VAR_INPUT
	in_max_Velo				: REAL;						(*	maximale Geschwindigkeit - Anwendereinheit z.B. xx mm/s *)
	in_Reglersperre			: BOOL;						(*  Software-Freigabe für die Achse  *)
	in_Freigabe				: BOOL;						(*  Freigabe JogMode und Positionieren *)
	in_Reset				: BOOL;						(*  Achs Reset  *)
	in_Hand					: BOOL;						(*  Handbetrieb  *)
	in_Auto					: BOOL;						(*  Automatikbetrieb  *)
	in_Auto_Override		: INT;						(*  in %  *)
	in_PosFenster			: REAL;						(*  Positionsfenster Achse in Position  *)
	in_Ref_pos				: REAL;						(*  Referenz-Wert der gesetzt werden soll  *)
	in_Bremse_PassQuitt		: BOOL;						(*	Passwort geschützes Bit aus der Visu zum Quittieren des Bremsentests, wenn der Test ..mal fehlgeschlagen ist	*)
	in_Endschalter_Min		: BOOL;						// AF - Reglerfreigabe für Fahrt negativ
	in_Endschalter_Max		: BOOL;						// AF - Reglerfreigabefür Fahrt positiv
	in_Normal_Drehmoment	: REAL := 100.0;			// AF - Drehmoment für den normalen Betrieb
END_VAR
VAR_OUTPUT
	out_ist_pos					: REAL;						(*  aktuelle ist Position  *)
	out_in_pos					: BOOL;						(*  Achse in Position (Soll=IST + - Positionsfenster) *)
	out_ziel_pos				: REAL;						(* aktuelle Zielposition *)
	out_nicht_ref				: BOOL;						(*  Achse ist nicht referenziert  *)
	out_bremse					: BOOL;						(*  Bremse lösen *)
	out_Achs_Status				: ST_AxisStatus;			(* 	aktueller Achsstatus *)
	out_Achs_Error				: BOOL;						(*  Achs Fehler *)
	out_Achs_ErrorID			: DINT;						(*  Achs Fehler ID *) 
	out_FB_Error				: BOOL;						(*  FB Fehler - intern *)
	out_FB_ErrorID				: DWORD;					(*  FB Fehler ID - intern *) 
	out_Bremsentest_Fehler		: BOOL;						(*	Bremsentestfehlerhaft *)
	out_Bremsentest_Fehler_3	: BOOL;						(*	Bremsentestfehlerhaft mehr als 3 mal fehlgeschlagen, Instandhalter informieren*)
	out_Bremsentest_Status		: DINT;						(*	0=alles ok, 1=Haltemoment zu gering, 2=Öffnungstest fehlerhaft, 3=...  *) 
	out_Bremsentest_notwendig	: BOOL;                       
	
END_VAR
VAR_IN_OUT
	inout_NC				: AXIS_REF;					(*  Schnittstelle zwischen der SPS und der NC  *)												
	inout_rexroth			: DUT_PD_InOut_Achsen;		(*  Schnittstelle zwischen der SPS und dem Regler  *)												
	inout_service			: DUT_Achse_Service;		(*  Eingangs-Variablen für den Servicebetrieb	 *)
	inout_Ref_start			: BOOL;						(*  Achse start referenzieren  *)
	inout_Auto_pos			: REAL;						(*  Auto Sollwert *)
	inout_Auto_start		: BOOL;						(*  Achse start Positionieren *)
	inout_Auto_stop			: BOOL;						(*  Achse stopp Positionieren *)
	inout_Bremsentest_Start	: BOOL;						(*	Bremsentest starten *)
END_VAR

VAR
	FB_ReadPos				: MC_ReadActualPosition;	(*  Aktuelle Istposition auslesen *)
	FB_ReadErrorID			: MC_ReadAxisError;			(*  FehlerID der Achse auslesen  *)
	FB_ReadStatus			: MC_ReadStatus;
	FB_POWER				: MC_POWER;					(*  Leistung ein-/ausschalten  *)
	FB_RESET				: MC_RESET;					(*  Achse resetten *)
	FB_Stop					: MC_Halt;					(*  Achse anhalten  *)
	FB_Jog					: MC_Jog;					(*  Achse tippen  *)
	FB_Move					: MC_MoveAbsolute;			(*  Achse positionieren  *)
	FB_Move_Seq_1			: MC_MoveAbsolute;
	FB_Move_Seq_2			: MC_MoveAbsolute;
	FB_Read_Parameter		: MC_ReadParameterSet;
	FB_Set_Position			: MC_SetPosition;
	FB_SoeReset				: Tc2_MC2_Drive.FB_SoEReset;
	start_seq				: BOOL;						(*  Start Merker Pos1<-> Pos 2 *)
	ton_verweil				: ton;
	ton_verzoegert			: tof;
	temp_in_pos_plus		: BOOL;
	temp_in_pos_minus		: BOOL;
	verz_reset				: ton;
	fl_start				: R_trig;					(* Start als Flanke auswerten und den Zähler erhöhen *)
	bremsentest_ver			: ton;						(* Verzögerungszeit zum Auswerten *)
	AnzahlVersuche			: INT;
	Achsparameter			: ST_AxisParameterSet;
END_VAR

// ***** Achs Status aktualisieren *******************************************************************************************
	//************************************************************************************************************************
	inout_NC();

	out_Achs_Status	:= FB_ReadStatus.Status;
	out_Achs_Error	:= FB_ReadErrorID.AxisErrorID > 0;

	IF out_Achs_Error 
		OR out_FB_Error
		OR in_reset
	THEN
		inout_Auto_start:=FALSE;
		inout_Auto_stop:=FALSE;
	END_IF
	
	if not inout_rexroth.S0145_steuerword.5 then
		inout_rexroth.S0092_drehmoment_grenzwert := REAL_TO_UINT(in_Normal_Drehmoment * 10);
	end_if
// ***** Aktuelle Zielposition ***********************************************************************************************
	//************************************************************************************************************************
	IF inout_nc.Status.Moving
	THEN
		out_ziel_pos := LREAL_TO_REAL(inout_NC.NcToPlc.TargetPos);
	ELSIF in_auto
		AND inout_auto_start
	THEN
		out_ziel_pos := inout_Auto_pos;
	ELSIF in_hand
		AND inout_service.betriebsart = 2				
			AND inout_service.plus_start
	THEN
		out_ziel_pos := inout_service.sollpos_hand;	
	END_IF	
	
// Freigabe positionieren ****************************************************************************************************
	//************************************************************************************************************************
	IF NOT in_Freigabe
	THEN
		inout_Auto_start 	:= FALSE;
		FB_Move.Execute		:= FALSE;
	END_IF	
	
// ***** Bremsentest starten *************************************************************************************************
	//************************************************************************************************************************
	out_Bremsentest_notwendig:= inout_rexroth.P0539_status_bremse.8; (* P-0-0539.8, Status Zeitintervall des Bremsentests  *)
	inout_rexroth.S0145_steuerword.2 := inout_Bremsentest_Start	(* P-0-0541, C2100 Kommando Haltesystemüberwachung *)
											AND inout_NC.Status.NotMoving;
	fl_start(clk:=inout_Bremsentest_Start);
	IF fl_start.q
	THEN
		AnzahlVersuche:=AnzahlVersuche+1;	
	END_IF
	
		// ***** Bremsentest Zeitverzögert auswerten *********************************************************************************	
			// ***********************************************************************************************************************
			bremsentest_ver(IN:=inout_rexroth.S0145_steuerword.2, pt:= T#4S);
			
		// ***** Bremsentest iO ******************************************************************************************************
			// ***********************************************************************************************************************
			IF bremsentest_ver.Q
				AND inout_rexroth.P0539_status_bremse.1 (* P-0-0539.1 - Status der Haltebremsenüberwachung *)
				AND inout_rexroth.P0539_status_bremse.2 (* P-0-0539.2 - Prüfstatus "Bremsenöffnung"  *)
				AND inout_rexroth.P0539_status_bremse.3 (* P-0-0539.3 - Prüfstatus "Haltemoment"  *)
			THEN
				inout_rexroth.S0145_steuerword.2:=FALSE;
				inout_Bremsentest_Start:=FALSE;
				AnzahlVersuche:=0;
				out_Bremsentest_Status:=0;
			END_IF
		// ***** Test niO und einen Fehler ausgeben ********************************************************************************** 
			// ***********************************************************************************************************************
			IF  bremsentest_ver.Q
					AND NOT inout_rexroth.P0539_status_bremse.2 (* P-0-0539.2 - Prüfstatus "Bremsenöffnung"  *)
			THEN
				out_Bremsentest_Status:=0;
				inout_Bremsentest_Start:=FALSE;
			END_IF
		
			IF  bremsentest_ver.Q
					AND NOT inout_rexroth.P0539_status_bremse.3 (* P-0-0539.3 - Prüfstatus "Haltemoment"  *)
			THEN
				out_Bremsentest_Status:=0;
				inout_Bremsentest_Start:=FALSE;
			END_IF
			
			IF out_Bremsentest_Status<>0
			THEN
				out_Bremsentest_Fehler:=TRUE;
				ELSE
					out_Bremsentest_Fehler:=FALSE;
			END_IF
		// ***** Quttierung nach einem Fehler ****************************************************************************************
			// ***********************************************************************************************************************
			IF AnzahlVersuche>=4
			THEN
				out_Bremsentest_Fehler_3:=TRUE;
			END_IF
			IF (in_Bremse_PassQuitt 
					OR (AnzahlVersuche<4))
				AND in_Reset
			THEN
				IF in_Bremse_PassQuitt
					AND AnzahlVersuche>=4  
				THEN
					AnzahlVersuche:=0;
				END_IF
				out_Bremsentest_Fehler_3:=FALSE;
				out_Bremsentest_Status:=0;
				inout_Bremsentest_Start:=FALSE;
			END_IF
		
// ***** Hand Betriebsart /Geschwindigkeit zurücksetzen***********************************************************************
	//************************************************************************************************************************
	IF NOT in_Hand
	THEN
		inout_service.betriebsart	:= 0;
		inout_service.override		:= 0;
	END_IF

// ***** Sollposition / Geschwindigkeit umkopieren ***************************************************************************
	//************************************************************************************************************************
	IF in_hand
	THEN
		FB_Move.Position		:= inout_service.sollpos_hand;
		FB_Power.Override		:= INT_TO_LREAL(inout_service.override);
		FB_Move.Velocity		:= in_max_velo;
		FB_Jog.Velocity			:= in_max_velo;
		fb_Move_seq_1.Velocity 	:= in_max_velo;
		fb_Move_seq_2.Velocity 	:= in_max_velo;
		fb_Move_seq_1.Position	:= inout_service.sollpos_hand;
		fb_Move_seq_2.Position	:= inout_service.pos_2;
		
		inout_rexroth.S0145_steuerword.5 := FALSE;
	ELSE
		FB_Move.Position		:= inout_Auto_pos;
		FB_Power.Override		:= INT_TO_LREAL(in_Auto_Override);
		FB_Move.Velocity		:= in_max_velo;
		FB_Jog.Velocity			:= 0.0;
	END_IF
	
	
// ***** Reset ***************************************************************************************************************
	//************************************************************************************************************************
	inout_rexroth.S0145_steuerword.0:=in_Reset;	// S-0-0099 - C0500 Reset Zustandsklasse 1 l

	FB_SoeReset(Axis := inout_NC, Execute := in_Reset OR FB_SoeReset.Busy);

	IF in_Reset
		AND (out_FB_Error
		OR out_Achs_Error) 
		OR ( in_Hand
				AND inout_service.betriebsart=0
				AND inout_service.minus_stop ) 
	THEN
		FB_Reset.Execute	:= inout_NC.NcToPlc.CoupleState <> 3; // Achse ist kein Slave
		FB_Stop.Execute		:= FALSE;
		FB_Move.Execute		:= FALSE;
		out_FB_Error		:= FALSE;
		out_FB_ErrorID		:= 0;
	END_IF

	verz_reset(	in:= FB_Reset.Execute,
				pt:= T#200MS);
	IF verz_reset.Q
	THEN
		FB_Reset.Execute := FALSE;
	END_IF

// ***** Achse stoppen *******************************************************************************************************
	//************************************************************************************************************************
	IF (in_Hand
			AND inout_service.minus_stop
			AND inout_service.betriebsart <> 1)
		OR inout_Auto_stop
		OR (NOT in_Freigabe
			AND inout_NC.Status.Moving
			AND inout_NC.NcToPlc.CoupleState <> 3) // Achse ist keine Slave Achse
		OR FB_Move.CommandAborted
		OR FB_Move.Error
		OR out_Achs_Error 
	THEN
		FB_STOP.Execute				:= TRUE;
		FB_Move.Execute				:= FALSE;
		start_seq 					:= FALSE;
		inout_service.plus_start 	:= FALSE;	
	END_IF                             
                                       
	IF (FB_STOP.Execute                
		AND FB_STOP.Done)              
	THEN                               
		inout_Auto_stop				:= FALSE;
		FB_STOP.Execute				:= FALSE;
		inout_service.minus_stop  	:= FALSE;
	END_IF

// ***** Referenzieren *******************************************************************************************************
	//************************************************************************************************************************
// Achse referenzieren - Absolutwert setzen
	inout_rexroth.S0052_ref_pos:=TRUNC(in_Ref_pos*10000.0);
	
	inout_rexroth.S0145_steuerword.1	:= NOT FB_Power.Enable
						AND ((in_Hand
								AND inout_service.betriebsart=4
								AND inout_service.plus_start)
							OR (in_Auto
								AND inout_Ref_start));

	IF inout_service.betriebsart=4
		AND (inout_rexroth.S0052_ref_pos = TRUNC(out_ist_pos*10000.0))
	THEN
		inout_service.plus_start:=FALSE;	
	END_IF
// ***** Achse positionieren *************************************************************************************************
	//************************************************************************************************************************
	IF ((in_Hand
			AND inout_service.betriebsart = 2				
			AND inout_service.plus_start)		
		OR (in_auto
			AND inout_Auto_start))
		AND NOT FB_Move.Done
		AND NOT FB_Move.busy
		AND NOT out_Achs_Error // optimierung 01.10.2020
		AND NOT out_Bremsentest_Fehler
		AND in_Freigabe
	THEN
		FB_Move.Execute:=TRUE;	
	END_IF

	IF (FB_Move.Execute
		AND FB_Move.Done)
		OR out_Achs_Error
	THEN
		FB_Move.Execute				:=FALSE;
		inout_Auto_start			:=FALSE;
		inout_service.plus_start 	:=FALSE;
	END_IF
	
	IF inout_service.betriebsart = 2
		AND (FB_Move.Execute
		AND FB_Move.Done)
	THEN 
		FB_Move.Execute := FALSE;
	END_IF
// ***** Handbetrieb - Achse POS1<->POS 2 ************************************************************************************
	//************************************************************************************************************************
	IF  in_hand
		AND inout_service.betriebsart = 3
		AND inout_service.plus_start
	THEN 
		start_seq := TRUE;
	END_IF

// ***** Handbetrieb - Achse tippen ******************************************************************************************
	//************************************************************************************************************************
	IF in_Hand
		AND inout_service.betriebsart=1
		AND NOT FB_Jog.CommandAborted
		AND NOT FB_Jog.Error
		AND NOT out_Bremsentest_Fehler
		AND in_Freigabe
	THEN
		FB_Jog.JogForward	:= inout_service.plus_start 
								AND inout_nc.NcToPlc.ActPos < (Achsparameter.fEncSoftEndMax - in_PosFenster);
		FB_Jog.JogBackwards	:= inout_service.minus_stop
								AND inout_nc.NcToPlc.ActPos > (Achsparameter.fEncSoftEndMin + in_PosFenster);
		
		// Geschwindigkeit tippen vor den Endlagen reduzieren
			// letzer 1% des Fahrwegs
		IF (FB_Jog.JogForward 
			AND inout_nc.NcToPlc.ActPos 
				> Achsparameter.fEncSoftEndMax - ((Achsparameter.fEncSoftEndMax - Achsparameter.fEncSoftEndMin) * 0.01))
			
			OR (FB_Jog.JogBackwards
				AND inout_nc.NcToPlc.ActPos  
					< Achsparameter.fEncSoftEndMin + ((Achsparameter.fEncSoftEndMax - Achsparameter.fEncSoftEndMin) * 0.01))
					
			AND FB_Power.Override > 5
		THEN
			FB_Power.Override := 5;
			
			// letzten 5% des Fahrwegs
		ELSIF (FB_Jog.JogForward 
			AND inout_nc.NcToPlc.ActPos 
				> Achsparameter.fEncSoftEndMax - ((Achsparameter.fEncSoftEndMax - Achsparameter.fEncSoftEndMin) * 0.05))
			
			OR (FB_Jog.JogBackwards
				AND inout_nc.NcToPlc.ActPos  
					< Achsparameter.fEncSoftEndMin + ((Achsparameter.fEncSoftEndMax - Achsparameter.fEncSoftEndMin) * 0.05))
					
			AND FB_Power.Override > 10	
		THEN
			FB_Power.Override := 10;
		END_IF
	ELSE
		FB_Jog.JogForward	:= FALSE;
		FB_Jog.JogBackwards	:= FALSE;
	END_IF
	
// ***** Aufruf der FB´s  ****************************************************************************************************
	//************************************************************************************************************************
	 ACT_Achse_NC_PTP();	
				
// ***** Bremse lösen ********************************************************************************************************
	//************************************************************************************************************************
	ton_verzoegert.IN 	:= FB_ReadStatus.Status.HasJob; 
	ton_verzoegert.pt 	:= T#2S;
	ton_verzoegert();
	out_bremse			:= ton_verzoegert.Q;
	
// ***** Achse in Position ***************************************************************************************************
	//************************************************************************************************************************
	out_in_pos := FB_ReadStatus.Status.InTargetPosition
					AND ((out_ist_pos >= (inout_Auto_pos - in_PosFenster))
					AND (out_ist_pos <= (inout_Auto_pos + in_PosFenster)));
					
// ***** Achse Referenzert ***************************************************************************************************
	//************************************************************************************************************************
	out_nicht_ref:=	 inout_rexroth.S0144_statusword.0;	//NOT FB_ReadStatus.Status.Homed;

// ***** FB Fehler auswerten und ausgeben ************************************************************************************
	//************************************************************************************************************************
	IF FB_Jog.Error
		AND FB_Jog.ErrorID > 0
	THEN
		out_FB_Error	:= TRUE;
		out_FB_ErrorID	:= FB_Jog.ErrorID;
		
	ELSIF FB_Move.Error
		AND FB_Move.ErrorID>0
	THEN
		FB_Move.Execute	:= FALSE;
		out_FB_Error	:= TRUE;
		out_FB_ErrorID	:= FB_Move.ErrorID;
		
	ELSIF FB_Stop.Error
		AND FB_Stop.ErrorID>0
	THEN	
		FB_Stop.Execute	:= FALSE;
		out_FB_Error	:= TRUE;
		out_FB_ErrorID	:= FB_Stop.ErrorID;
		
	ELSIF FB_Reset.Error
		AND FB_Reset.ErrorID>0
	THEN
		FB_Reset.Execute	:= FALSE;
		out_FB_Error		:= TRUE;
		out_FB_ErrorID		:= FB_Reset.ErrorID;
	END_IF			

					
// ***** Servicetasten zurück setzen ************************************************************************************
	//************************************************************************************************************************
	IF inout_service.betriebsart <> 1
		AND inout_service.betriebsart <> 4
	THEN
		inout_service.plus_start := FALSE;				
		inout_service.minus_stop := FALSE;				
	END_IF
	
	inout_Auto_start := FALSE;

ACTION ACT_Achse_NC_PTP:
	
	FB_ReadErrorID(	Axis:=inout_NC,
					Enable:=TRUE,
					AxisErrorID=>);
	out_achs_ErrorID:= DWORD_TO_DINT(FB_ReadErrorID.AxisErrorID);	
	
	
	FB_ReadPos(		Axis:=inout_NC,
					Enable:=TRUE,
					Position=> ,
					Position=> );				
				
	out_ist_pos:=inout_service.istpos:=LREAL_TO_REAL(FB_ReadPos.Position);
	
	FB_Read_Parameter(	Parameter:= Achsparameter, 
						Axis:= inout_NC, 
						Execute:= in_Reglersperre, 
						Done=> , 
						Busy=> , 
						Error=> , 
						ErrorID=> );
			
	FB_ReadStatus(	Axis:=inout_NC,
					Enable:=TRUE);
				
	FB_Power.Enable:=in_Reglersperre AND (inout_service.betriebsart<>4	OR inout_ref_start);	
	FB_Power.Enable_Negative := FB_Power.Enable AND in_Endschalter_Min;
	FB_Power.Enable_Positive :=	FB_Power.Enable	AND in_Endschalter_Max;
				
	FB_Power(	Axis:=inout_NC,
				Enable:=,
				Enable_Positive:=,
				Enable_Negative:=,
				Override:=,
				BufferMode:=MC_Aborting,
				Options:=	);
				
	FB_Reset(	Axis:=inout_NC,
				Execute:=	);
				
	FB_Stop(	Axis:=inout_NC,
				Execute:=,
				Deceleration:=0,				(* Bei einem Wert von 0 wirkt die mit dem letzten Move-Kommando parametrierte Verzögerung *)
				Jerk:=0,						(* Bei einem Wert von 0 wirkt der mit dem letzten Move-Kommando parametrierte Ruck *)		
				BufferMode:= MC_Aborting);		 // Wichtig !!!!				
																		
	FB_Move(	Axis:=inout_NC,
				Execute:=,
				Position:=,
				Velocity:=,
				Acceleration:=0,				(* Beschleunigung, bei einem Wert von 0 wirkt die Standardbeschleunigung aus der Achskonfiguration im System Manager *)
				Deceleration:=0,				(* Verzögerung, bei einem Wert von 0 wirkt die Standardverzögerung aus der Achskonfiguration im System Manager *)
				Jerk:=0, 						(* Ruck, bei einem Wert von 0 wirkt der Standardruck aus der Achskonfiguration im System Manager *)
				BufferMode:= MC_Buffered);		
									
	FB_Jog(		Axis:=inout_NC,
				JogForward:=,
				JogBackwards:=,
				Mode:= MC_JOGMODE_STANDARD_SLOW, //MC_JOGMODE_CONTINOUS,
				Position:=,						(* nicht in diesem Mode notwendig *)
				Velocity:=,
				Acceleration:=0,				(* Beschleunigung, bei einem Wert von 0 wirkt die Standardbeschleunigung aus der Achskonfiguration im System Manager *)
				Deceleration:=0,				(* Verzögerung, bei einem Wert von 0 wirkt die Standardverzögerung aus der Achskonfiguration im System Manager *)
				Jerk:=0 );						(* Ruck, bei einem Wert von 0 wirkt der Standardruck aus der Achskonfiguration im System Manager *)

	
	ton_verweil(in:= (NOT fb_move_seq_1.active 
						AND NOT fb_move_seq_2.active
						AND inout_service.betriebsart=3),
				pt:= INT_TO_TIME(inout_service.zeit));
				
	FB_Move_Seq_1(
				Execute:= 	(start_seq 
								AND NOT fb_move_seq_2.busy 
								AND ton_verweil.Q),
				Position:= 			,
				Velocity:= 			,
				Acceleration:= ,				(* Beschleunigung, bei einem Wert von 0 wirkt die Standardbeschleunigung aus der Achskonfiguration im System Manager *)
				Deceleration:= ,			 	(* Verzögerung, bei einem Wert von 0 wirkt die Standardverzögerung aus der Achskonfiguration im System Manager *)
				Jerk:=,							(* Ruck, bei einem Wert von 0 wirkt der Standardruck aus der Achskonfiguration im System Manager *) 
				BufferMode:= MC_Buffered,
				Options:= ,
				Axis:=inout_NC,
				Done=>				,
				Busy=> 				,
				Active=> 			,
				CommandAborted=> 	,
				Error=> 			,
				ErrorID=> 			);


	FB_Move_Seq_2(
				Execute:= 		(start_seq	
								AND fb_move_seq_1.done
								AND ton_verweil.Q),
				Position:= 		,
				Velocity:= 			,
				Acceleration:= ,				(* Beschleunigung, bei einem Wert von 0 wirkt die Standardbeschleunigung aus der Achskonfiguration im System Manager *)
				Deceleration:= ,				(* Verzögerung, bei einem Wert von 0 wirkt die Standardverzögerung aus der Achskonfiguration im System Manager *)
				Jerk:= ,						(* Ruck, bei einem Wert von 0 wirkt der Standardruck aus der Achskonfiguration im System Manager *)
				BufferMode:= MC_Buffered,
				Options:= ,
				Axis:= inout_NC,
				Done=>				,
				Busy=> 				,
				Active=> 			,
				CommandAborted=> 	,
				Error=> 			,
				ErrorID=> 			);
END_ACTION

METHOD M_AutoPos : BOOL
VAR_INPUT
	SollPos		:REAL;
END_VAR
	
	// Drehmomentgrenze deaktivieren
	inout_rexroth.S0145_steuerword.5 := FALSE;

	if not inout_rexroth.S0144_statusword.6 then
		FB_Move.Options.IgnorePositionMonitoring := false;
		
		inout_Auto_pos := SollPos;
		inout_Auto_start := TRUE;
	
		IF out_in_pos 
		AND Func_InRange(IstPos := inout_NC.NcToPlc.ActPos, SollPos := inout_Auto_pos, Fenster := in_PosFenster) 
		THEN
			M_AutoPos := TRUE;
		END_IF 
		
	end_if
END_METHOD

METHOD M_AutoTorque : BOOL
VAR_INPUT
	SollPos	: REAL;
	Torque	: REAL;  // Prozentwert
END_VAR
	
	inout_rexroth.S0145_steuerword.5 := TRUE;
	if inout_rexroth.S0144_statusword.6 then
		FB_Move.Options.IgnorePositionMonitoring := true;
		inout_rexroth.S0092_drehmoment_grenzwert := REAL_TO_UINT(Torque * 10);
	
		inout_Auto_pos := SollPos;
		inout_Auto_start := TRUE;
	
		IF (out_in_pos 
		AND Func_InRange(IstPos := inout_NC.NcToPlc.ActPos, SollPos := inout_Auto_pos, Fenster := in_PosFenster))
		OR inout_rexroth.S0144_statusword.5
		THEN
			M_AutoTorque := TRUE;
		END_IF 
	
	end_if
END_METHOD

END_FUNCTION_BLOCK

// ---- SRT_Allgemein/0010_Bausteine_mitDuts/POUs/Servos_NC/FB_MasterSlaveSpeedControl.TcPOU
FUNCTION_BLOCK FB_MasterSlaveSpeedControl
VAR_INPUT
	SpeedMaster	:REAL;
	SpeedSlave1	:REAL;
	SpeedSlave2	:REAL;
	SpeedSlave3	:REAL;
	hysterese	:REAL;
	
END_VAR
VAR_OUTPUT
	speedMasterSlave_OK :BOOL;
END_VAR
VAR
	speedSlave1_OK	:BOOL;
	speedSlave2_OK	:BOOL;
	speedSlave3_OK	:BOOL;
END_VAR

IF SpeedSlave1 < SpeedMaster + hysterese
	AND SpeedSlave1 > SpeedMaster - hysterese
THEN
	speedSlave1_OK :=TRUE;
ELSE
	speedSlave1_OK :=FALSE;
END_IF

IF SpeedSlave2 < SpeedMaster + hysterese
	AND SpeedSlave2 > SpeedMaster - hysterese
THEN
	speedSlave2_OK :=TRUE;
ELSE
	speedSlave2_OK :=FALSE;
END_IF

IF SpeedSlave3 < SpeedMaster + hysterese
	AND SpeedSlave3 > SpeedMaster - hysterese
THEN
	speedSlave3_OK :=TRUE;
ELSE
	speedSlave3_OK :=FALSE;
END_IF


IF speedSlave1_OK
	AND speedSlave2_OK
	AND speedSlave3_OK
	AND speedMaster>0
THEN
	speedMasterSlave_ok := TRUE;
ELSE
	speedMasterSlave_ok := FALSE;
END_IF

END_FUNCTION_BLOCK

// ---- SRT_Allgemein/0010_Bausteine_mitDuts/POUs/Servos_NC/FB_Nc_Kanal.TcPOU
FUNCTION_BLOCK FB_Nc_Kanal
(*
	Ansteuerung eines NC-Kanals 
	Autor O.E.
	Erstellt 13.01.2022
	Version 1.0 	
*)
VAR_INPUT
	in_Kanal_Id						:UDINT;					(* NC Kanal Nummer *)
	in_Gruppe_Id					:UDINT;					(* NC Gruppennummer *)
	in_X_Id							:UDINT;					(* X-Achs Id *)
	in_Y_Id							:UDINT;					(* Y-Achs Id *)
	in_Z_Id							:UDINT;					(* Z-Achs Id *)
	in_Pfad							:STRING[80];			(* Pfad wo das NC-Programm liegr *)
	in_PName						:STRING[80];			(* Name des zubearbeitenden NC-Programms *)
	in_Override						:DINT;					(* Gesamt Override der bearbeitung 0-100%*)
	in_NcToPlc						:NCTOPLC_NCICHANNEL_REF;
END_VAR

VAR_OUTPUT
	out_PlcToNc						:PLCTONC_NCICHANNEL_REF;
	out_P_uebernommen				:BOOL;					(* vorgegebenes Programm übernommen soll=ist *)
	out_FBErr						:BOOL;
	out_FBErrId						:UDINT;
END_VAR

VAR_IN_OUT
	inout_NcReset					:BOOL;				(* Kanal Reset *)
	inout_NcGruppe_koppeln			:BOOL;				(* Achsen zu einer Gruppe zusammen fügen *)
	inout_NcStart					:BOOL;				(* NC-Ablauf starten *)
	inout_NcStopOverrideNull		:BOOL;				(* NC-Ablauf unterbrechen -Override=0 *)
	inout_NcEinzelsatzStart			:BOOL;				(* NC-Ablauf im Einzelsatzbetrieb abarbeiten *)
	inout_NcEinzelsatzWeiter		:BOOL;				(* nächster Satz *)
	inout_NcStatus					:Dut_Nc_Kanal;
	
END_VAR

VAR
	                    	
	AxTo3D			 				:CfgBuildExt3dGroup;
	AxToPTP							:CfgReconfigGroup;
	AxTo3DLoad						:BOOL;
	AxToPTPLoad						:BOOL;                  		
                            	
	Einzel							:ItpsingleBlock;
	EinzelChange					:BOOL;
	EinzelStart						:R_Trig;
	EinzelStop						:f_Trig;
	ProgAnw							:ItpLoadProgEx;
	ProgStart						:ItpStartStopEx;
	ProgReset						:ItpResetEx;
                    			
	PLoad							:BOOL;
	
	FlPGrd							:R_TRIG;
	FlPBearb						:R_TRIG;
	Pfad_PNr 	 					:STRING[80];
	FlPReset						:R_Trig;
                    	    	
	TStart							:TON;
	PStart							:R_TRIG;
                    				
	OverInit						:BOOL;
                   				
	MFuncTime						:TON;
    MFuncQuitt						:ItpResetFastMFuncEx;  
	MFuncConfirm					:ItpConfirmHsk;
	FlMFuncNoReq					:r_trig;

	PName_akt:						STRING[80];
	
	PBearb:							BOOL;
	Override						:DINT;
	Start:							BOOL;
	Stop:							BOOL;
	Untbr:							BOOL;
	Reset:							BOOL;

	 
END_VAR

//***** Info zum NCI-Ablauf *************************************************************************************
	//**********************************************************************************************************
(*
	1. Einzelachsen fehlerfrei in Grundposition
	2. Gruppe bilden / Achsen koppeln			-> CfgBuildExt3dGroup
	3. Interpreter Reset						-> ItpResetEx
	4. Programm laden							-> ItpLoadProgEx
	5. Einzelsatzbetrieb (optinal)				-> ItpSingleBlock
	6. Programm starten							-> ItpStartStopEx
	7. Warten auf M-Funktion und quittieren		-> PLCTONC_NCICHANNEL_REF.MFuncGranted
		M-Funktion steht an							-> ItpIsHskMFunc
		M_FunktionsNummer							-> ItpGetHskMFunc
	8. Gruppe auflösen / Achsen entkoppeln		-> CfgReconfigGroup
*)
//***** Kanalreset *********************************************************************************************
	//**********************************************************************************************************
	Reset:= inout_NcReset;

//***** Achsen Config ******************************************************************************************
	//**********************************************************************************************************

		IF inout_NcGruppe_koppeln
		THEN
			IF NOT inout_NcStatus.AxTo3DOk
			AND NOT AxTo3D.bErr
			THEN
				AxTo3DLoad:= TRUE;
				inout_NcStatus.AxToPTPOk:= FALSE;
			END_IF;
		ELSE
			IF NOT inout_NcStatus.AxToPTPOk
			AND NOT AxToPTP.bErr
			THEN
				AxToPTPLoad:= TRUE;
				inout_NcStatus.AxTo3DOk:= FALSE;
			END_IF;
		END_IF;

	// Achsen in 3D Gruppe uebergeben 
	AxTo3D	(	nGroupId		:=in_Gruppe_Id,
				nXAxisId		:=in_X_Id,
				nYAxisId		:=in_Y_Id,
				nZAxisId		:=in_Z_Id,
				nQ1AxisId		:=0,
				nQ2AxisId		:=0,
				nQ3AxisId		:=0,
				nQ4AxisId		:=0,
				nQ5AxisId		:=0,
				bExecute		:=AxTo3DLoad,
				tTimeOuT		:=T#1S,				
				bErr			=>,
				nErrId			=>,);


	IF AxTo3D.bBusy THEN
		inout_NcStatus.AxTo3Dok	:= TRUE;
		AxTo3DLoad			:= FALSE;
	END_IF;

	IF AxTo3D.bErr THEN
		inout_NcStatus.AxTo3Dok	:= FALSE;
	END_IF;

	// Achsen zurueck in PTP 
	AxToPTP(nGroupId		:=in_Gruppe_Id,
			bExecute		:=AxToPTPLoad,
			tTimeOuT		:=T#1S);

	IF AxToPTP.bBusy THEN
		inout_NcStatus.AxToPTPok	:= TRUE;
		AxToPTPLoad			:= FALSE;
	END_IF;

	IF AxToPTP.bErr THEN
		inout_NcStatus.AxToPTPok	:= FALSE;
	END_IF;
	
//***** Aktuelles NC-Programm laden ***************************************************************************
	//**********************************************************************************************************
	PName_akt		:=DWORD_TO_STRING (in_NcToPlc.LoadedProg);
	
	// NC-Programm laden 
	IF in_PName <> PName_akt
		AND NOT Reset
		AND NOT ProgAnw.bBusy 
		AND in_PName <>''
	THEN
		PLoad:=TRUE;
		ELSE
			PLoad:=FALSE;
	END_IF;

	Pfad_PNr := CONCAT (in_Pfad, in_PName) ;
	Pfad_PNr := CONCAT (Pfad_PNr,'.NC') ;

	ProgAnw (sNciToPlc	:=in_NcToPlc,
			sPrg		:=Pfad_PNr,
			nLength		:=INT_TO_UDINT((LEN(Pfad_PNr))),
			bExecute	:=PLoad,
			tTimeOuT	:=T#10S,				
			bErr		=>,
			nErrId		=>);

	IF ProgAnw.bBusy 
	THEN
		PLoad			:= FALSE;
	END_IF;

	// Ueberpruefung Grundstellung / Bearbeitungsprogramm geladen 
	PBearb	:=(in_PName = PName_akt);
	// Nach dem laden des Programmes muß ein Reset durchgefuehrt werden 
	FlPBearb (CLK:=PBearb);

	IF FlPGrd.Q
	OR FlPBearb.Q
	THEN
		Reset:= TRUE;
	END_IF;

	out_P_uebernommen:= in_PName = PName_akt;
//***** NC Err *************************************************************************************************
	//**********************************************************************************************************
	inout_NcStatus.Err	:=  in_NcToPlc.ItpState= Tc2_NCI.NCI_INTERPRETER_ABORTED
					 OR in_NcToPlc.ErrorCode<> 0;

//***** NC Aktiv ***********************************************************************************************
	//**********************************************************************************************************
	inout_NcStatus.Aktiv	:= in_NcToPlc.ItpState > Tc2_NCI.NCI_INTERPRETER_READY
					AND NOT inout_NcStatus.Err;

//***** NC Ready ***********************************************************************************************
	//**********************************************************************************************************
	IF in_NcToPlc.ItpState = Tc2_NCI.NCI_INTERPRETER_READY
	THEN
		inout_NcStatus.Ready:= TRUE;
	END_IF

	IF in_NcToPlc.ItpState = Tc2_NCI.NCI_INTERPRETER_IDLE
		OR inout_NcStatus.Err
		OR inout_NcStatus.Aktiv
	THEN
		inout_NcStatus.Ready:= FALSE;
	END_IF
//***** NC Run *************************************************************************************************
	//**********************************************************************************************************
	inout_NcStatus.Run	:= in_NcToPlc.ItpState = Tc2_NCI.NCI_INTERPRETER_RUNNING;
				
//***** Einzelsatzbetrieb **************************************************************************************
	//**********************************************************************************************************
	EinzelStart(clk:=inout_NcEinzelsatzStart);
	EinzelStop(clk:=inout_NcEinzelsatzStart);
	
	IF EinzelStart.q 
		AND NOT inout_NcStart
		AND in_NcToPlc.ItpState = Tc2_NCI.NCI_INTERPRETER_READY
	THEN
		//  ItpSingleBlockOff   	:= 0 		-> Einzelsatz aus
		//	ItpSingleBlockNck   	:= 1 		-> Einzelsatz im NC-Kern
		//	ItpSingleBlockIntp  	:= 16#4000	-> Einzelsatz im Interpreter
		Einzel.nMode:= ItpSingleBlockIntp  ;
		EinzelChange:=TRUE;
	END_IF

	IF EinzelStop.Q
	THEN 
		Einzel.nMode:=ItpSingleBlockOff;
		EinzelChange:=TRUE;
	END_IF
		
	Einzel(sNciToPlc			:= in_NcToPlc,
			bExecuteModeChange	:= EinzelChange,
			bTriggerNext		:= inout_NcEinzelsatzWeiter);
		
	IF Einzel.bBusy
	THEN
		EinzelChange:=FALSE;
	END_IF	
//***** NC Start/Stop Programm *********************************************************************************
	//**********************************************************************************************************
	TStart.IN	:=inout_NcStart 
					AND inout_NcStatus.AxTo3DOk
					AND NOT EinzelChange;
	TStart(PT	:=T#50ms);

	PStart (CLK:=TStart.Q);

	IF PStart.Q
	THEN
		Start:=TRUE;
	END_IF

	IF NOT  inout_NcStart
		OR 	inout_NcStatus.Aktiv
	THEN
		Start:=FALSE;
	END_IF 

	IF NOT inout_NcGruppe_koppeln
		AND in_NcToPlc.ItpState = Tc2_NCI.NCI_INTERPRETER_RUNNING
	THEN
		Stop:=TRUE;
		Reset:=TRUE;
	END_IF


	IF in_NcToPlc.ItpState <> Tc2_NCI.NCI_INTERPRETER_RUNNING
	THEN
		Stop:=FALSE;
	END_IF

	ProgStart(sNciToPlc		:=in_NcToPlc,
				bStart		:=Start,
				bStop		:=Stop,
				tTimeOut	:=T#1S,				
				bErr		=>,
				nErrId		=>);

	IF ProgStart.bBusy
	THEN
		Start:= FALSE;
		Stop:= FALSE;
	END_IF;

//***** NC Reset Programm **************************************************************************************
	//**********************************************************************************************************
	IF  in_NcToPlc.ItpState = Tc2_NCI.NCI_INTERPRETER_READY
		AND in_NcToPlc.ErrorCode = 0
	THEN
		Reset:= FALSE;
	END_IF;

	ProgReset(nChnId	:=in_Kanal_Id,
				nGrpId	:=in_Gruppe_Id,	
				bExecute:=Reset,
				tTimeOut:=T#1S,				
				bErr		=>,
				nErrId		=>);

	Reset:= FALSE;

//***** Kanal Override *****************************************************************************************
	//**********************************************************************************************************
	IF NOT OverInit
	THEN
		in_Override	:=1000000;	(* Init 100% *)
		OverInit	:=TRUE;
	ELSE
		Override:=in_Override*10000;
	END_IF;

	out_PlcToNc.ChnAxesOvr 		:=DINT_TO_UDINT(Override);

	Untbr					:=inout_NcStopOverrideNull;

	IF Untbr
	THEN
		out_PlcToNc.ChnAxesOvr:=0; (* 0% *)
	END_IF;

//***** M-Befehle **********************************************************************************************
	//**********************************************************************************************************
	inout_NcStatus.MFuncReq:=ItpIsHskMFunc(in_NcToPlc);
	inout_NcStatus.MFuncNr:=ItpGetHskMFunc(in_NcToPlc);
	 
 
	MFuncTime(IN:=(inout_NcStatus.MFuncReq), PT:=T#100MS);

	IF MFuncTime.Q
		AND inout_NcStatus.MFuncQuitt 
		AND (inout_NcStatus.MFuncNr=inout_NcStatus.MFuncQuittNr)
	THEN
		out_PlcToNc.MFuncGranted:=1;
		ELSE
			out_PlcToNc.MFuncGranted:=0;			
	END_IF

	FlMFuncNoReq(clk:=NOT inout_NcStatus.MFuncReq);															
	IF FlMFuncNoReq.Q
	THEN  		
		inout_NcStatus.MFuncQuitt:=FALSE;														
	END_IF
	
//***** Fehler ausgeben ****************************************************************************************
	//**********************************************************************************************************

	IF ProgAnw.bErr
	THEN
		out_FBErr:=TRUE;
		out_FBErrId:=ProgAnw.nErrId;
	END_IF
	
	IF ProgStart.bErr
	THEN
		out_FBErr:=TRUE;
		out_FBErrId:=ProgStart.nErrId;
	END_IF

	IF AxTo3D.bErr
	THEN
		out_FBErr:=TRUE;
		out_FBErrId:=AxTo3D.nErrId;
	END_IF

	IF AxToPTP.bErr
	THEN
		out_FBErr:=TRUE;
		out_FBErrId:=AxToPTP.nErrId;
	END_IF

	IF ProgReset.bErr
	THEN
		out_FBErr:=TRUE;
		out_FBErrId:=ProgReset.nErrId;
	END_IF
	
//*****************************************************************************************************
	//**********************************************************************************************************
	FlPReset(clk:=in_NcToPlc.ItpState = Tc2_NCI.NCI_INTERPRETER_READY);
	IF FlPReset.Q
		OR inout_NcReset
	THEN
		inout_NcGruppe_koppeln			:=
		inout_NcStart					:=
		inout_NcStopOverrideNull		:=
		inout_NcEinzelsatzStart			:=
		inout_NcEinzelsatzWeiter		:=
		inout_NcStatus.MFuncQuitt		:=FALSE;
		inout_NcStatus.MFuncQuittNr		:=0;
	
		IF NOT ProgAnw.bErr
			AND NOT ProgStart.bErr
			AND NOT AxTo3D.bErr
			AND NOT AxToPTP.bErr
			AND NOT ProgReset.bErr
		THEN
			out_FBErr					:=FALSE;
			out_FBErrId					:=0;
		END_IF

			inout_NcReset				:=FALSE;		
		
	END_IF

END_FUNCTION_BLOCK

// ---- SRT_Allgemein/0010_Bausteine_mitDuts/POUs/Zaehler/FB_Laufzeit.TcPOU
FUNCTION_BLOCK FB_Laufzeit
VAR_INPUT
    inAktiv				: BOOL;		(* Betriebsstatus, 1 = aktiv, 0 = inaktiv *)
END_VAR

VAR_OUTPUT
    outLetzeteLaufzeit	: REAL;		(* letzte Laufzeit in Sekunden *)	
END_VAR

VAR_IN_OUT
    inoutGesamtLaufzeit	: REAL;		(* Gesamt Laufzeit in Minuten *)	
END_VAR

VAR
	t500msAn			: ton;
	t500msAus			: tof;
	t500ms				: BOOL;
	fl_start			: r_trig;
	fl_stop				: f_trig;
	zaehler				: UDINT;
END_VAR

(* Blinktakt *)
	t500msAn(IN:=NOT t500msAus.Q , PT:=T#500MS);
	t500msAus(IN:=t500msAn.Q , PT:=T#500MS , Q=>t500ms);
	
(* Start *)
	fl_start(CLK:=t500ms AND inAktiv);
	IF fl_start.Q
	THEN
		zaehler:=zaehler+1;
	END_IF
	
(* Zählwert auswertent *)
	fl_stop(CLK:=inAktiv);
	IF fl_stop.Q
	THEN
		outLetzeteLaufzeit:=	TO_REAL (zaehler);
		inoutGesamtLaufzeit:= 	inoutGesamtLaufzeit + (TO_REAL (zaehler)/60);
	END_IF

(* Initialisierung des internen Zählers *)
	IF NOT inAktiv
	THEN
		zaehler:=0;
	END_IF

END_FUNCTION_BLOCK

// ---- SRT_Allgemein/0010_Bausteine_mitDuts/POUs/Zaehler/FB_SpindelInBearbeitung.TcPOU
FUNCTION_BLOCK FB_SpindelInBearbeitung
VAR_INPUT
	inStart				:BOOL;	
	inAktiveSpindeln	:ARRAY[1..16] OF BOOL; 		// aktive Spindeln im Bohrvorgang
END_VAR
VAR_IN_OUT
	inoutSpindel		:ARRAY[1..16] OF UDINT; 	// Anzahl wie oft eine Spindel benutzt wurde
END_VAR
VAR
	a					: INT:=1;
	fl_start			: r_trig;	
END_VAR

	fl_start(CLK:=inStart);
	IF fl_start.Q
	THEN
		FOR a:=1 TO 16 DO
			IF inAktiveSpindeln[a]
			THEN
				inoutSpindel[a]:=inoutSpindel[a]+1;
			END_IF
		END_FOR		
	END_IF

END_FUNCTION_BLOCK

// ---- SRT_Allgemein/Bus/Busdiagnose.TcPOU
FUNCTION_BLOCK Busdiagnose
VAR_INPUT
			
	
END_VAR
VAR_OUTPUT
	
END_VAR
VAR_IN_OUT
Bus:DUT_Busdiagnose;
END_VAR
VAR
{attribute 'tc_no_symbol'}
StatesLesen : FB_ecGetAllSlaveStates;
{attribute 'tc_no_symbol'}
AddressenLesen : FB_EcGetConfSlaves;
{attribute 'tc_no_symbol'}
TopologieLesen: FB_EcGetSlaveTopologyInfo;
{attribute 'tc_no_symbol'}
AnzahlEtherCatDevices: FB_EcGetSlaveCount;
{attribute 'tc_no_symbol'}
Slaveslesen: FB_EcGetScannedSlaves;
{attribute 'tc_no_symbol'}
States	 : ARRAY [0..ec_Max_Slaves] OF ST_EcSlaveState;
{attribute 'tc_no_symbol'}
StatesAlt	 : ARRAY [0..ec_Max_Slaves] OF ST_EcSlaveState;
{attribute 'tc_no_symbol'}
Config	 : ARRAY [0..ec_Max_Slaves] OF ST_EcSlaveConfigData;
{attribute 'tc_no_symbol'}
Topology	 : ARRAY [0..ec_Max_Slaves] OF ST_TopologyDataEx;
{attribute 'tc_no_symbol'}
Slaves	 : ARRAY [0..ec_Max_Slaves] OF ST_EcSlaveScannedData;
{attribute 'tc_no_symbol'}
lesen :BOOL;
{attribute 'tc_no_symbol'}

{attribute 'tc_no_symbol'}
busy:BOOL;
{attribute 'tc_no_symbol'}
error:BOOL;
{attribute 'tc_no_symbol'}
errorId: UDINT;
{attribute 'tc_no_symbol'}
Slave: UINT;

{attribute 'tc_no_symbol'}	
busy2:BOOL;
{attribute 'tc_no_symbol'}
error2:BOOL;
{attribute 'tc_no_symbol'}
errorID2: UDINT;
{attribute 'tc_no_symbol'}
Slaves2: UINT;

{attribute 'tc_no_symbol'}	
busy3:BOOL;
{attribute 'tc_no_symbol'}
error3:BOOL;
{attribute 'tc_no_symbol'}
errorID3: UDINT;
{attribute 'tc_no_symbol'}
Slaves3: UINT;

{attribute 'tc_no_symbol'}	
busy4:BOOL;
{attribute 'tc_no_symbol'}
error4:BOOL;
{attribute 'tc_no_symbol'}
errorID4: UDINT;
{attribute 'tc_no_symbol'}
Slaves4: UINT;

{attribute 'tc_no_symbol'}	
busy5:BOOL;
{attribute 'tc_no_symbol'}
error5:BOOL;
{attribute 'tc_no_symbol'}
errorID5: UDINT;
{attribute 'tc_no_symbol'}
Slaves5: UINT;

{attribute 'tc_no_symbol'}	
zyklen : INT;
{attribute 'tc_no_symbol'}
i: UDINT;
{attribute 'tc_no_symbol'}	
AnzahlFehler :UINT;
END_VAR



AnzahlEtherCatDevices(
	sNetId:= F_CreateAmsNetId(nIds:=  bus.AmsNetId), 
	bExecute:= lesen, 
	tTimeout:=T#500MS , 
	bBusy=> busy4 , 
	bError=> error4, 
	nErrId=>errorID4 , 
	nSlaves=> Bus.AnzahlTeilnehmer);

StatesLesen(
	sNetId:= F_CreateAmsNetId(nIds:=  bus.AmsNetId),
	pStateBuf:= ADR(States), 
	cbBufLen:= SIZEOF(States), 
	bExecute:= lesen, 
	tTimeout:= T#500MS, 
	bBusy=>busy , 
	bError=> error, 
	nErrId=> errorId, 
	nSlaves=> Slave
 );
 
 AddressenLesen(
	sNetId:=F_CreateAmsNetId(nIds:=  bus.AmsNetId), 
	pArrEcConfSlaveInfo:= ADR(Config) , 
	cbBufLen:= SIZEOF(Config), 
	bExecute:= lesen, 
	tTimeout:=  T#500MS, 
	bBusy=> busy2, 
	bError=> error2,
	nErrorId=> errorID2, 
	nSlaves=> Slaves2);
	
TopologieLesen(
	sNetId:= F_CreateAmsNetId(nIds:=  bus.AmsNetId), 
	pAddrBuf:= ADR(Topology) , 
	cbBufLen:= SIZEOF(Topology), 
	bExecute:= lesen, 
	tTimeout:= T#500MS, 
	bBusy=> busy3, 
	bError=> error3,
	nErrId=> errorID3, 
	nSlaves=> Slaves3);
	
	Slaveslesen(sNetId:= F_CreateAmsNetId(nIds:=  bus.AmsNetId), 
	pArrEcScannedSlaveInfo := ADR(slaves) , 
	cbBufLen:= SIZEOF(slaves), 
	bExecute:= lesen, 
	tTimeout:= T#500MS, 
	bBusy=> busy5, 
	bError=> error5,
	nErrorId=> errorID5, 
	nSlaves=> Slaves5);
	
	zyklen := zyklen + 1;
	
	IF zyklen >= 100 THEN
		zyklen := 0;
		lesen := NOT lesen;
	END_IF
	
	IF Bus.AnzahlTeilnehmer > SIZEOF(Bus.Daten) THEN
		Bus.AnzahlTeilnehmer := SIZEOF(Bus.Daten);
		END_IF
		
	IF  Bus.AnzahlTeilnehmer > 0 AND lesen AND Config[0].sType <> ''
AND NOT busy
AND NOT busy2
AND NOT busy3
AND NOT busy4
//AND NOT busy5

 THEN
		FOR i := 0 TO  Bus.AnzahlTeilnehmer-1 DO
			
			Bus.Daten[i].adresse := Config[i].nAddr;
			Bus.Daten[i].deviceState := States[i].deviceState;
			Bus.Daten[i].linkState := States[i].linkState;
			Bus.Daten[i].Name := Config[i].sName;
			Bus.Daten[i].PortA := Topology[i].stPhysicalAddr.portA;
			Bus.Daten[i].PortB := Topology[i].stPhysicalAddr.portB;
			Bus.Daten[i].PortC := Topology[i].stPhysicalAddr.portC;
			Bus.Daten[i].PortD := Topology[i].stPhysicalAddr.portD;
			Bus.Daten[i].productCode := Config[i].stSlaveIdentity.productCode;
			Bus.Daten[i].revisionNo := Config[i].stSlaveIdentity.revisionNo;
			Bus.Daten[i].serialnNo := Config[i].stSlaveIdentity.serialNo;
			Bus.Daten[i].Typ := Config[i].nDevType;
			Bus.Daten[i].TypName := Config[i].sType;
			
		END_FOR
	

	FOR i := 0 TO  Bus.AnzahlTeilnehmer-1 DO
		IF States[i].deviceState <> StatesAlt[i].deviceState
			OR States[i].linkState <> StatesAlt[i].linkState
			THEN
			IF Bus.Update = 100 THEN
				Bus.Update :=0;
			ELSE				
				Bus.Update :=Bus.Update+ 1;
				EXIT;
			END_IF	
		END_IF			
	END_FOR
	
	AnzahlFehler := 0;
	FOR i := 0 TO  Bus.AnzahlTeilnehmer-1 DO
		StatesAlt[i].deviceState := States[i].deviceState;
			StatesAlt[i].linkState := States[i].linkState;
			IF StatesAlt[i].deviceState <> 8 //OR StatesAlt[i].linkState <> 36
				THEN
					AnzahlFehler := AnzahlFehler + 1;
					
			END_IF		
	END_FOR
	//Bus.AnzahlFehler := Bus.AnzahlFehler - 234;
	IF AnzahlFehler <=0 THEN
		AnzahlFehler := 0;
		ELSE
			AnzahlFehler := AnzahlFehler ;//-233;
		END_IF
	END_IF
	bus.AnzahlFehler := AnzahlFehler;
Bus.FehlerfreiAktiv := NOT error AND NOT error2 AND NOT error3 AND NOT error4;

END_FUNCTION_BLOCK
